// TIA Portal V17 export
// export: Created 2022-07-28T18:02:50.8696399Z, ExportSetting None, DisplayName Totally Integrated Automation Portal, DisplayVersion V17, DisplayName TIA Portal Openness, DisplayVersion V17, DisplayName TIA Portal Teamcenter Gateway, DisplayVersion V17, DisplayName TIA Portal Version Control Interface, DisplayVersion V17, DisplayName TIA Portal Test Suite Advanced, DisplayVersion V17, DisplayName SINAMICS Startdrive Advanced, DisplayVersion V17, DisplayName SINAMICS DCC, DisplayVersion V17, DisplayName SINAMICS Startdrive G130, G150, S120, S150, SINAMICS MV, S210, DisplayVersion V17, DisplayName SINAMICS Startdrive G110M, G120, G120C, G120D, G120P, G115D, DisplayVersion V17, DisplayName STEP 7 Professional, DisplayVersion V17, DisplayName SIMATIC Energy Suite, DisplayVersion V17, DisplayName STEP 7 CFC, DisplayVersion V17, DisplayName STEP 7 Safety, DisplayVersion V17, DisplayName WinCC Advanced / Unified PC, DisplayVersion V17, DisplayName SIMATIC Visualization Architect, DisplayVersion V17
FUNCTION_BLOCK "Lib_FB_AnalogFlowmeter"   // FB7, SCL
{ S7_Optimized_Access := 'TRUE' }
AUTHOR : bean
// Analog sensor functional block
// stored: AutoNumber false, MemoryReserve 100, SetENOAutomatically false
   VAR_INPUT
      I_Initialization { ExternalAccessible := 'False'; ExternalVisible := 'False'; ExternalWritable := 'False'} : Bool := FALSE;   // 1 = Restart PLC is active (First scan)
      IR_Raw { ExternalAccessible := 'False'; ExternalVisible := 'False'; ExternalWritable := 'False'} : Real;   // Sensor input
      IR_High { ExternalAccessible := 'False'; ExternalVisible := 'False'; ExternalWritable := 'False'} : Real := 27648.0;   // Max sensor input val, PLC unit
      IR_Low { ExternalAccessible := 'False'; ExternalVisible := 'False'; ExternalWritable := 'False'} : Real;   // Min sensor input val, PLC unit
      IR_Coef { ExternalAccessible := 'False'; ExternalVisible := 'False'; ExternalWritable := 'False'} : Real := 60.0;   // Coeffitient for convert flow to unit/min (t/h -> kg/min ) by dividing
      II_Mode { ExternalAccessible := 'False'; ExternalVisible := 'False'; ExternalWritable := 'False'} : Int := -1;   // 0 - analog;
      I_GlobalRST { ExternalAccessible := 'False'; ExternalVisible := 'False'; ExternalWritable := 'False'} : Bool;   // Reset faults
      I_Puls_1s { ExternalAccessible := 'False'; ExternalVisible := 'False'; ExternalWritable := 'False'} : Bool;   // 1 = Once per 1 sec
      IR_CycleTime { ExternalAccessible := 'False'; ExternalVisible := 'False'; ExternalWritable := 'False'} : Real;   // PLC last cycle time
      II_Obj_ID { ExternalAccessible := 'False'; ExternalVisible := 'False'; ExternalWritable := 'False'} : Int := -1;   // Tech ID of object
   END_VAR
   VAR_OUTPUT
      QR_ScalledVal { ExternalAccessible := 'False'; ExternalVisible := 'False'; ExternalWritable := 'False'} : Real;   // Output scaled sensor value
      Q_HH { ExternalAccessible := 'False'; ExternalVisible := 'False'; ExternalWritable := 'False'} : Bool;   // High level Alarm
      Q_H { ExternalAccessible := 'False'; ExternalVisible := 'False'; ExternalWritable := 'False'} : Bool;   // High level Warning
      Q_L { ExternalAccessible := 'False'; ExternalVisible := 'False'; ExternalWritable := 'False'} : Bool;   // Low level Warning
      Q_LL { ExternalAccessible := 'False'; ExternalVisible := 'False'; ExternalWritable := 'False'} : Bool;   // Low level Alarm
      Q_Overshoot { ExternalAccessible := 'False'; ExternalVisible := 'False'; ExternalWritable := 'False'} : Bool;   // Sensor value overshoot
      Q_BadSensor { ExternalAccessible := 'False'; ExternalVisible := 'False'; ExternalWritable := 'False'} : Bool;   // Sensor in zero
      Q_DBReadErr { ExternalAccessible := 'False'; ExternalVisible := 'False'; ExternalWritable := 'False'} : Bool;   // Object DB reading fault
   END_VAR
   VAR_IN_OUT
      IQ_PLC_CycleInfo : Variant;
   END_VAR
   VAR
      s_SimMode { ExternalAccessible := 'False'; ExternalVisible := 'False'; ExternalWritable := 'False'} : Bool;   // Simulation mode is active
      s_FltCondition_HH { ExternalAccessible := 'False'; ExternalVisible := 'False'; ExternalWritable := 'False'} : Bool;   // Condition for high level fault
      s_FltCondition_H { ExternalAccessible := 'False'; ExternalVisible := 'False'; ExternalWritable := 'False'} : Bool;   // Condition for high level warning
      s_FltCondition_L { ExternalAccessible := 'False'; ExternalVisible := 'False'; ExternalWritable := 'False'} : Bool;   // Condition for low level warning
      s_FltCondition_LL { ExternalAccessible := 'False'; ExternalVisible := 'False'; ExternalWritable := 'False'} : Bool;   // Condition for low level fault
      s_Flt_HH { ExternalAccessible := 'False'; ExternalVisible := 'False'; ExternalWritable := 'False'} : Bool;
      s_Flt_LL { ExternalAccessible := 'False'; ExternalVisible := 'False'; ExternalWritable := 'False'} : Bool;
      slr_CurrentFlow_u_s { ExternalAccessible := 'False'; ExternalVisible := 'False'; ExternalWritable := 'False'} : LReal;   // Current flow in unit/sec
      slr_PrevFlow_u_s { ExternalAccessible := 'False'; ExternalVisible := 'False'; ExternalWritable := 'False'} : LReal;   // Previous flow in unit/sec
      slr_CountFlow_min { ExternalAccessible := 'False'; ExternalVisible := 'False'; ExternalWritable := 'False'} : LReal;
      slr_FlowMid_min { ExternalAccessible := 'False'; ExternalVisible := 'False'; ExternalWritable := 'False'} : LReal;
      si_CountTimePoints { ExternalAccessible := 'False'; ExternalVisible := 'False'; ExternalWritable := 'False'} : Int;
      slr_Count_unit { ExternalAccessible := 'False'; ExternalVisible := 'False'; ExternalWritable := 'False'} : LReal;   // Counter for units
      s_Enable { ExternalAccessible := 'False'; ExternalVisible := 'False'; ExternalWritable := 'False'} : Struct   // Enable/disable faults detection
         HH : Bool := true;   // High fault
         H : Bool := true;   // High warning
         L : Bool := true;   // Low warning
         LL : Bool := true;   // Low fault
      END_STRUCT;
      s_Suppressed { ExternalAccessible := 'False'; ExternalVisible := 'False'; ExternalWritable := 'False'} : Struct   // Suppress faults
         HH : Bool;   // High fault
         H : Bool;   // High warning
         L : Bool;   // Low warning
         LL : Bool;   // Low fault
      END_STRUCT;
      s_TON_HH { ExternalAccessible := 'False'; ExternalVisible := 'False'; ExternalWritable := 'False'} : "Lib_FB_Timer_ON_Simple";
      s_TON_H { ExternalAccessible := 'False'; ExternalVisible := 'False'; ExternalWritable := 'False'} : "Lib_FB_Timer_ON_Simple";
      s_TON_L { ExternalAccessible := 'False'; ExternalVisible := 'False'; ExternalWritable := 'False'} : "Lib_FB_Timer_ON_Simple";
      s_TON_LL { ExternalAccessible := 'False'; ExternalVisible := 'False'; ExternalWritable := 'False'} : "Lib_FB_Timer_ON_Simple";
      s_EdgeError { ExternalAccessible := 'False'; ExternalVisible := 'False'; ExternalWritable := 'False'} : "Lib_FB_Edge";
      s_EdgeWarning { ExternalAccessible := 'False'; ExternalVisible := 'False'; ExternalWritable := 'False'} : "Lib_FB_Edge";
      s_EdgeOvershot { ExternalAccessible := 'False'; ExternalVisible := 'False'; ExternalWritable := 'False'} : "Lib_FB_Edge";
   END_VAR
   VAR RETAIN
      s_Simulation { ExternalAccessible := 'False'; ExternalVisible := 'False'; ExternalWritable := 'False'} : Struct
         Obj_DATA_BACKUP : Struct
            Config : "_AnalogFlowmeter_Config";
            s_Enable : Struct   // Enable/disable faults detection
               HH : Bool := true;   // High fault
               H : Bool := true;   // High warning
               L : Bool := true;   // Low warning
               LL : Bool := true;   // Low fault
            END_STRUCT;
            s_Suppressed : Struct   // Suppress faults
               HH : Bool;   // High fault
               H : Bool;   // High warning
               L : Bool;   // Low warning
               LL : Bool;   // Low fault
            END_STRUCT;
         END_STRUCT;
      END_STRUCT;
      s_Obj_Retain_BUp { ExternalAccessible := 'False'; ExternalVisible := 'False'; ExternalWritable := 'False'} : Struct
         Config : "_AnalogFlowmeter_Config";
         s_Enable : Struct   // Enable/disable faults detection
            HH : Bool := true;   // High fault
            H : Bool := true;   // High warning
            L : Bool := true;   // Low warning
            LL : Bool := true;   // Low fault
         END_STRUCT;
         s_Suppressed : Struct   // Suppress faults
            HH : Bool;   // High fault
            H : Bool;   // High warning
            L : Bool;   // Low warning
            LL : Bool;   // Low fault
         END_STRUCT;
      END_STRUCT;
   END_VAR
   VAR_TEMP
      t_SomeFault : Bool;
      t_SomeWarning : Bool;
      t_SensorOvershoot : Bool;
      t_Flt_HH : Bool;
      t_Flt_H : Bool;
      t_Flt_L : Bool;
      t_Flt_LL : Bool;
      t_Flt_SensMax : Bool;
      t_Flt_SensMin : Bool;
      t_ExclFlt : Bool;   // Excluded (suppressed) fault is active
      t_RST_FLT : Bool;
      t_DBReadErr : Bool;   // Fault while DB reading
      t_ResetCurrCnt : Bool;   // 1 = Reset current counter
      t_ResetGenCnt : Bool;   // 1 = Reset general counter
      ti_DBReadErr : Int;   // Fault # while DB reading
      ti_CMDLogic : Int;   // Command word for logic
      tlr_CntLastCycle : LReal;   // Counter by last cycle, unit
      t_WholeRange : Bool;
      t_WholeRangeP : Bool;
      ti_NumObjDB : UInt;   // Number of DB for storage object data
      t_ObjAny_HMI : DB_ANY;   // Ref to object data
      t_ObjVar_HMI : Variant;   // Ref to object data
      t_ObjAny_PLC : DB_ANY;   // Ref to object data
      t_ObjVar_PLC : Variant;   // Ref to object data
      tr_OutVal : Real;   // Output Sensor Value
      tr_OutValSens : Real;   // Output value in sensor range
      tr_OutValSensProc : Real;   // Output value in sensor range in %
      tr_CurrMaxRange : Real;   // Current maxixmum value of the range
      tr_CurrMinRange : Real;   // Current minimum value of the range
      tr_SP_HH : Real;
      tr_SP_H : Real;
      tr_SP_L : Real;
      tr_SP_LL : Real;
      tr_DeltaFlt : Real;
      tr_SensorVal : Real;
      tlr_Frac_CntU : LReal;   // Frac from unit counter
      tlr_CoefChecked : LReal;
      tui_IntPart_CntU : UDInt;   // Integer part from unit counter
      td_DB_ShiftHMI : DInt;   // Object DB number shift
      td_DB_ShiftPLC : DInt;   // Object DB number shift
      t_PLC_CycleInfo : "Lib_PLC_CycleInfo";
      t_Obj_HMI : "lib_udt_AnalogFlowmeter_HMI";
      t_Obj_PLC : "lib_udt_AnalogFlowmeter_PLC";
      t_InternalData : "Lib_UDT_Int";   // Internal data
   END_VAR
BEGIN
   REGION Inputs
       //Global reset to logic
       #t_RST_FLT := #I_GlobalRST;

       //Set internal data
       REGION Internal data
           #t_InternalData.AlwTrue := true;
           #t_InternalData.AlwFalse := false;
           #t_InternalData.i_Alw0 := 0;
           #t_InternalData.b_Alw0 := b#16#0;
           #t_InternalData.w_Alw0 := w#16#0;
           #t_InternalData.d_Alw0 := dw#16#0;
       END_REGION

       //Reinit tempory variables
       REGION Reinit tempory variables
           #t_WholeRange := false;
           #t_WholeRangeP := false;
           #t_ResetCurrCnt := false;
           #t_ResetGenCnt := false;
           #tr_SP_HH := 90.0;
           #tr_SP_H := 80.0;
           #tr_SP_L := 20.0;
           #tr_SP_LL := 10.0;
           #tr_DeltaFlt := 2.0;

       END_REGION

       //Read data  PLC 
       VariantGet(SRC := #IQ_PLC_CycleInfo,
                  DST => #t_PLC_CycleInfo);

       //Read Object data
       //Reinit temp values
       #t_Obj_HMI := "D_ZeroTypes".AnalogFlowmeter_HMI;
       #t_Obj_PLC := "D_ZeroTypes".AnalogFlowmeter_PLC;
       #td_DB_ShiftHMI := "D_General_ProgramDATA".ui_Shift_DBSens_HMI;
       #td_DB_ShiftPLC := "D_General_ProgramDATA".ui_Shift_DBSens_PLC;

       IF #II_Obj_ID >= 0
       THEN
           //Read HMI data
           #ti_NumObjDB := DINT_TO_UINT(INT_TO_DINT(#II_Obj_ID) + #td_DB_ShiftHMI);
           #t_ObjAny_HMI := UINT_TO_DB_ANY(#ti_NumObjDB);
           #t_ObjVar_HMI := DB_ANY_TO_VARIANT(in := #t_ObjAny_HMI, err => #ti_DBReadErr);

           //If DB exist and convertion without error
           IF #ti_DBReadErr = 0
           THEN
               VariantGet(SRC := #t_ObjVar_HMI,
                          DST => #t_Obj_HMI);
           ELSE
               #t_DBReadErr := true;
           END_IF;

           //Read PLC data
           #ti_NumObjDB := DINT_TO_UINT(INT_TO_DINT(#II_Obj_ID) + #td_DB_ShiftPLC);
           #t_ObjAny_PLC := UINT_TO_DB_ANY(#ti_NumObjDB);
           #t_ObjVar_PLC := DB_ANY_TO_VARIANT(in := #t_ObjAny_PLC, err => #ti_DBReadErr);

           //If DB exist and convertion without error
           IF #ti_DBReadErr = 0
           THEN
               VariantGet(SRC := #t_ObjVar_PLC,
                          DST => #t_Obj_PLC);
           ELSE
               #t_DBReadErr := true;
           END_IF;
       ELSE
           #t_DBReadErr := true;
       END_IF;

       //Read retain data if initialization is active
       IF #I_Initialization
       THEN
           #t_Obj_HMI.Config := #s_Obj_Retain_BUp.Config;
           #s_Enable := #s_Obj_Retain_BUp.s_Enable;
           #s_Suppressed := #s_Obj_Retain_BUp.s_Suppressed;

           #slr_PrevFlow_u_s := 0.0;
           #slr_Count_unit := 0.0;
           #slr_CountFlow_min := 0.0;
           #slr_FlowMid_min := 0.0;
           #si_CountTimePoints := 0;
       END_IF;

       //Define CMD by priority
       IF #t_PLC_CycleInfo.CMD_GLOBAL <> 0
       THEN
           #ti_CMDLogic := #t_PLC_CycleInfo.CMD_GLOBAL;
       ELSE
           IF #t_Obj_HMI.CMD <> 0
           THEN
               #ti_CMDLogic := #t_Obj_HMI.CMD;
               #t_Obj_HMI.CMD := 0;
           END_IF;
       END_IF;

       CASE #ti_CMDLogic OF
           0:  //Do nothing
               ;
           7:  //Sim mode ON
               IF NOT #s_SimMode
               THEN
                   #s_SimMode := TRUE;
                   #s_Simulation.Obj_DATA_BACKUP.Config := #t_Obj_HMI.Config;
                   #s_Simulation.Obj_DATA_BACKUP.s_Enable := #s_Enable;
                   #s_Simulation.Obj_DATA_BACKUP.s_Suppressed := #s_Suppressed;
               END_IF;

           8:  //Sim mode OFF
               IF #s_SimMode
               THEN
                   #s_SimMode := FALSE;
                   #t_Obj_HMI.Config := #s_Simulation.Obj_DATA_BACKUP.Config;
                   #s_Enable := #s_Simulation.Obj_DATA_BACKUP.s_Enable;
                   #s_Suppressed := #s_Simulation.Obj_DATA_BACKUP.s_Suppressed;
               END_IF;

           31..32://Reset faults
               #t_RST_FLT := TRUE;
           76:  //Display whole range
               #t_Obj_HMI.Config.i_HMI_SensValRange := 0;
           77:  //Display whole range, %
               #t_Obj_HMI.Config.i_HMI_SensValRange := 1;
               (* IF #II_Mode <> 0 THEN
                   #t_Obj_HMI.Config.i_HMI_SensValRange := 1;
               ELSE
                   #t_Obj_HMI.Config.i_HMI_SensValRange := 0;
               END_IF; *)(*
           78:  //Display a part of range
               #t_Obj_HMI.Config.i_HMI_SensValRange := 2;
           79:  //Display a part of range, %
               #t_Obj_HMI.Config.i_HMI_SensValRange := 3; *)
           60: //HH fault enable / disable
               #s_Enable.HH := NOT #s_Enable.HH;
           61: //H fault enable / disable
               #s_Enable.H := NOT #s_Enable.H;
           62: //L fault enable / disable
               #s_Enable.L := NOT #s_Enable.L;
           63: //LL fault enable / disable
               #s_Enable.LL := NOT #s_Enable.LL;
           64: //HH fault suppressed / consider
               #s_Suppressed.HH := NOT #s_Suppressed.HH;
           65: //H fault suppressed / consider
               #s_Suppressed.H := NOT #s_Suppressed.H;
           66: //L fault suppressed / consider
               #s_Suppressed.L := NOT #s_Suppressed.L;
           67: //LL fault suppressed / consider
               #s_Suppressed.LL := NOT #s_Suppressed.LL;
           500: //Reset current counter
               #t_ResetCurrCnt := true;
           501: //Reset general counter
               #t_ResetGenCnt := true;
           ELSE//
               ;
       END_CASE;

       CASE #t_Obj_HMI.Config.i_HMI_SensValRange OF
           0..1:  //Valid range
               ;
           ELSE  //Invalid range
               #t_Obj_HMI.Config.i_HMI_SensValRange := 1;
       END_CASE;

       #tr_SensorVal := #IR_Raw;
   END_REGION

   REGION Min/max values check
       //Start reading limits, offset and setpoints --------limits-offset-setpoints--------limits-offset-setpoints
       //            ************
       IF #t_Obj_HMI.Config.r_MinVal > #t_Obj_HMI.Config.r_MaxVal THEN
           #t_Obj_HMI.Config.r_MinVal := #t_Obj_HMI.Config.r_MaxVal;
       END_IF;
   END_REGION

   REGION Calculate percentage value depending on the mode of the sensor

       CASE #II_Mode OF
           0:  //Analog input like 0 - 27648 -> 0 - 75 C
               IF (#IR_High - #IR_Low) <> 0.0
               THEN
                   #tr_OutValSensProc := (#tr_SensorVal - #IR_Low) / (#IR_High - #IR_Low) * 100.0;
               ELSE
                   #tr_OutValSensProc := 0.0;
               END_IF;

           ELSE  //Undefined or unchoiced type of the sensor
               #t_Obj_HMI := "D_ZeroTypes".AnalogFlowmeter_HMI;
               #t_Obj_PLC := "D_ZeroTypes".AnalogFlowmeter_PLC;

               //Write Object data
               //DB num 
               IF #II_Obj_ID >= 0
                   AND NOT #t_DBReadErr
               THEN
                   //Write HMI data
                   VariantPut(SRC := #t_Obj_HMI,
                              DST := #t_ObjVar_HMI);

                   //Write PLC data
                   VariantPut(SRC := #t_Obj_PLC,
                              DST := #t_ObjVar_PLC);
               ELSE
                   #t_DBReadErr := true;
               END_IF;

               #QR_ScalledVal := 0.0;
               #Q_HH :=
               #Q_H :=
               #Q_L :=
               #Q_LL :=
               #Q_Overshoot :=
               #Q_DBReadErr := false;

               RETURN;
       END_CASE;

       //Calculate all others out values
       #tr_OutValSens := (#t_Obj_HMI.Config.r_MaxVal - #t_Obj_HMI.Config.r_MinVal) * #tr_OutValSensProc / 100.0 + #t_Obj_HMI.Config.r_MinVal;

       //Assign display mode depending by display mode
       CASE #t_Obj_HMI.Config.i_HMI_SensValRange OF
           0: //Display whole range
               #tr_OutVal := #tr_OutValSens + #t_Obj_HMI.Config.r_Offset;
               #tr_CurrMaxRange := #t_Obj_HMI.Config.r_MaxVal;
               #tr_CurrMinRange := #t_Obj_HMI.Config.r_MinVal;
               #t_WholeRange := true;
           1: //Display whole range (percents)
               #tr_OutVal := #tr_OutValSensProc + #t_Obj_HMI.Config.r_Offset;
               #tr_CurrMaxRange := 100.0;
               #tr_CurrMinRange := 0.0;
               #t_WholeRangeP := true;
           ELSE
               ;
       END_CASE;

       REGION Check limits, zero of sensor ect.
           IF #tr_SensorVal < #IR_Low
               OR #tr_SensorVal > #IR_High
           THEN
               #t_SensorOvershoot := true;
           END_IF;

           IF #tr_OutValSensProc < -5.0
           THEN
               #t_Flt_SensMin := TRUE;
               #tr_OutVal := 0.0;
           END_IF;

           IF #tr_OutValSensProc > 105.0
           THEN
               #t_Flt_SensMax := TRUE;
               #tr_OutVal := 0.0;
           END_IF;

           IF #tr_OutVal > #tr_CurrMaxRange
           THEN
               #tr_OutVal := #tr_CurrMaxRange;
           END_IF;
           IF #tr_OutVal < #tr_CurrMinRange
           THEN
               #tr_OutVal := #tr_CurrMinRange;
           END_IF;
       END_REGION

       IF #s_SimMode
       THEN
           #tr_OutVal := #t_Obj_HMI.Config.r_DisplayData;
           #tr_OutValSens := #t_Obj_HMI.Config.r_DisplayData;
       END_IF;

   END_REGION

   REGION Calculate counters by flow
       //Reset counters
       IF #t_ResetCurrCnt
       THEN
           #t_Obj_HMI.Config.r_CountCurr := 0;
       END_IF;
       IF #t_ResetGenCnt
       THEN
           #t_Obj_HMI.Config.r_CountGen := 0;
       END_IF;

       IF #I_Puls_1s
       THEN

           //Check coeffitient
           IF #IR_Coef <> 0.0
           THEN
               #tlr_CoefChecked := REAL_TO_LREAL(#IR_Coef);
           ELSE
               #tlr_CoefChecked := 1.0;
           END_IF;

           //Calculate counter by previous cycle
           #slr_CurrentFlow_u_s := REAL_TO_LREAL(#tr_OutValSens) / #tlr_CoefChecked;

           //Count time points and sum of flow
           #slr_CountFlow_min += #slr_CurrentFlow_u_s;
           #si_CountTimePoints += 1;

           IF #si_CountTimePoints >= 60
           THEN
               #slr_FlowMid_min += #slr_CountFlow_min / 60.0;

               #si_CountTimePoints := 0;

               #tui_IntPart_CntU := DINT_TO_UDINT(TRUNC(#slr_FlowMid_min));
               #tlr_Frac_CntU := FRAC(#slr_FlowMid_min);
               #slr_CountFlow_min := 0.0;//#tlr_Frac_CntU;
               #slr_FlowMid_min := #tlr_Frac_CntU;

               #t_Obj_HMI.Config.r_CountCurr += #tui_IntPart_CntU;
               #t_Obj_HMI.Config.r_CountGen += #tui_IntPart_CntU;
               #t_Obj_HMI.Config.r_CountHour += #tui_IntPart_CntU;
           END_IF;

       END_IF;


   END_REGION

   REGION Setpoints values check
       //            ************
       IF #t_Obj_HMI.Config.r_LL_Setpoint < #tr_CurrMinRange
       THEN
           #t_Obj_HMI.Config.r_LL_Setpoint := #tr_CurrMinRange;
       ELSIF #t_Obj_HMI.Config.r_LL_Setpoint > #tr_CurrMaxRange
       THEN
           #t_Obj_HMI.Config.r_LL_Setpoint := #tr_CurrMaxRange;
       END_IF;

       IF #t_Obj_HMI.Config.r_HH_Setpoint > #tr_CurrMaxRange
       THEN
           #t_Obj_HMI.Config.r_HH_Setpoint := #tr_CurrMaxRange;
       ELSIF #t_Obj_HMI.Config.r_HH_Setpoint < #tr_CurrMinRange
       THEN
           #t_Obj_HMI.Config.r_HH_Setpoint := #tr_CurrMinRange;
       END_IF;
       //            ************
       IF #t_Obj_HMI.Config.r_H_Setpoint > #t_Obj_HMI.Config.r_HH_Setpoint
       THEN
           #t_Obj_HMI.Config.r_H_Setpoint := #t_Obj_HMI.Config.r_HH_Setpoint;
       ELSIF #t_Obj_HMI.Config.r_H_Setpoint < #t_Obj_HMI.Config.r_LL_Setpoint
       THEN
           #t_Obj_HMI.Config.r_H_Setpoint := #t_Obj_HMI.Config.r_LL_Setpoint;
       END_IF;

       IF #t_Obj_HMI.Config.r_L_Setpoint > #t_Obj_HMI.Config.r_H_Setpoint
       THEN
           #t_Obj_HMI.Config.r_L_Setpoint := #t_Obj_HMI.Config.r_H_Setpoint;
       ELSIF #t_Obj_HMI.Config.r_L_Setpoint < #t_Obj_HMI.Config.r_LL_Setpoint
       THEN
           #t_Obj_HMI.Config.r_L_Setpoint := #t_Obj_HMI.Config.r_LL_Setpoint;
       END_IF;

       //            ************         
       #tr_SP_HH := #t_Obj_HMI.Config.r_HH_Setpoint;
       #tr_SP_H := #t_Obj_HMI.Config.r_H_Setpoint;
       #tr_SP_L := #t_Obj_HMI.Config.r_L_Setpoint;
       #tr_SP_LL := #t_Obj_HMI.Config.r_LL_Setpoint;
       #tr_DeltaFlt := #t_Obj_HMI.Config.r_Hysteresis;
       //Finish reading limits, offset and setpoints --------limits-offset-setpoints--------limits-offset-setpoints
   END_REGION

   REGION Warnings AND faults

       REGION Setpoints intersection    
           //Setpoints intersection
           IF #tr_SP_HH <= #tr_CurrMaxRange
               AND #tr_SP_H <= #tr_CurrMaxRange
           THEN
               #s_FltCondition_HH := (#tr_SP_HH <= #tr_OutVal)
               OR (#s_FltCondition_HH
               AND #tr_OutVal >= (#tr_SP_HH - #tr_DeltaFlt));

               #s_FltCondition_H := (#tr_SP_H <= #tr_OutVal)
               OR (#s_FltCondition_H
               AND #tr_OutVal >= (#tr_SP_H - #tr_DeltaFlt));

           ELSE
               #s_FltCondition_HH := FALSE;
               #s_FltCondition_H := FALSE;
           END_IF;

           IF #tr_SP_LL >=  #tr_CurrMinRange
               AND #tr_SP_L >= #tr_CurrMinRange
           THEN
               #s_FltCondition_LL := (#tr_SP_LL >= #tr_OutVal)
               OR (#s_FltCondition_LL
               AND #tr_OutVal <= (#tr_SP_LL + #tr_DeltaFlt));

               #s_FltCondition_L := (#tr_SP_L >= #tr_OutVal)
               OR (#s_FltCondition_L
               AND #tr_OutVal <= (#tr_SP_L + #tr_DeltaFlt));
           ELSE
               #s_FltCondition_LL := FALSE;
               #s_FltCondition_L := FALSE;
           END_IF;
       END_REGION

       //Enabled faults and warnings check
       #s_FltCondition_HH := #s_FltCondition_HH AND #s_Enable.HH;
       #s_FltCondition_H := #s_FltCondition_H AND #s_Enable.H;
       #s_FltCondition_L := #s_FltCondition_L AND #s_Enable.L;
       #s_FltCondition_LL := #s_FltCondition_LL AND #s_Enable.LL;

       #s_TON_HH(IB_StartTimerInput := #s_FltCondition_HH,
               IR_CycleTime := #IR_CycleTime,
               IR_SpTime := #t_Obj_HMI.Config.r_WarnDetectTime);

       #s_TON_H(IB_StartTimerInput := #s_FltCondition_H,
              IR_CycleTime := #IR_CycleTime,
              IR_SpTime := #t_Obj_HMI.Config.r_WarnDetectTime);

       #s_TON_L(IB_StartTimerInput := #s_FltCondition_L,
              IR_CycleTime := #IR_CycleTime,
              IR_SpTime := #t_Obj_HMI.Config.r_WarnDetectTime);

       #s_TON_LL(IB_StartTimerInput := #s_FltCondition_LL,
               IR_CycleTime := #IR_CycleTime,
               IR_SpTime := #t_Obj_HMI.Config.r_WarnDetectTime);

       #t_Flt_HH := #s_TON_HH.QB_TimerOut AND NOT #s_Suppressed.HH;
       #t_Flt_H := #s_TON_H.QB_TimerOut AND NOT #s_Suppressed.H;
       #t_Flt_L := #s_TON_L.QB_TimerOut AND NOT #s_Suppressed.L;
       #t_Flt_LL := #s_TON_LL.QB_TimerOut AND NOT #s_Suppressed.LL;

       //Excluded (suppressed) fault is active
       #t_ExclFlt := (#s_TON_HH.QB_TimerOut AND #s_Suppressed.HH)
       OR (#s_TON_H.QB_TimerOut AND #s_Suppressed.H)
       OR (#s_TON_L.QB_TimerOut AND #s_Suppressed.L)
       OR (#s_TON_LL.QB_TimerOut AND #s_Suppressed.LL)
       ;

       #s_Flt_HH := #t_Flt_HH
       OR (#s_Flt_HH
       AND NOT #t_RST_FLT);

       #s_Flt_LL := #t_Flt_LL
       OR (#s_Flt_LL
       AND NOT #t_RST_FLT);


       //Some fault is active
       #t_SomeFault := #s_Flt_HH
       OR #s_Flt_LL
       ;
       //Some warning is active
       #t_SomeWarning := #t_Flt_H
       OR #t_Flt_L
       ;
       //New fault checking
       #s_EdgeError(IB_Input := #t_SomeFault);

       //New warning checking
       #s_EdgeWarning(IB_Input := #t_SomeWarning);

       //New overshot detected
       #s_EdgeOvershot(IB_Input := #t_SensorOvershoot
                       OR #t_Flt_SensMax
                       OR #t_Flt_SensMin);
   END_REGION

   REGION PLC State + Counter
       "Lib_FC_ASens_CycleInfo_Count_State"(Alarm := #t_SomeFault,
                                            AlarmNew := #s_EdgeError.QB_EdgePos,
                                            Warning := #t_SomeWarning,
                                            WarningNew := #s_EdgeWarning.QB_EdgePos,

                                            ErrorBad := #t_SensorOvershoot
                                            OR #t_Flt_SensMax
                                            OR #t_Flt_SensMin,
                                            ErrorBadNew := #s_EdgeOvershot.QB_EdgePos,
                                            Simulation := #s_SimMode,
                                            PLC_CycleInfo := #t_PLC_CycleInfo);
   END_REGION

   REGION BUp Data
       IF NOT #I_Initialization
       THEN
           #s_Obj_Retain_BUp.Config := #t_Obj_HMI.Config;
           #s_Obj_Retain_BUp.s_Enable := #s_Enable;
           #s_Obj_Retain_BUp.s_Suppressed:= #s_Suppressed;
       END_IF;
   END_REGION

   REGION Outputs
       //Outputs
       //Object DBs
       //HMI DB
       #t_Obj_HMI.Config.r_DisplayData := #tr_OutVal;
       #t_Obj_HMI.ID := #II_Obj_ID;
       #t_Obj_HMI.CLSID := 40;
       #t_Obj_HMI.Status.r_HW_Value := #IR_Raw;

       //Alarm word
       #t_Obj_HMI.Status.w_AW1.%X0 := #s_Flt_HH;           //x0 - HH fault is active                       
       #t_Obj_HMI.Status.w_AW1.%X1 := #t_Flt_H;            //x1 - H fault is active                        
       #t_Obj_HMI.Status.w_AW1.%X2 := #t_Flt_L;            //x2 - L fault is active                        
       #t_Obj_HMI.Status.w_AW1.%X3 := #s_Flt_LL;           //x3 - LL fault is active                       
       #t_Obj_HMI.Status.w_AW1.%X4 := #t_SensorOvershoot;  //x4 - Overshoot is active (act val > Maxlim)   
       #t_Obj_HMI.Status.w_AW1.%X5 := #t_Flt_SensMax;      //x5 - Exceeding the maximum                    
       #t_Obj_HMI.Status.w_AW1.%X6 := #t_Flt_SensMin;      //x6 - Exceeding the minimum                    
       #t_Obj_HMI.Status.w_AW1.%X7 := #s_SimMode;          //x7 - Sim mode is active                       
       #t_Obj_HMI.Status.w_AW1.%X8 := NOT #s_SimMode;      //x8 - Sim mode disabled
   (*    #t_Obj_HMI.Status.w_AW1.%X9     := ;    //x9 - 
       #t_Obj_HMI.Status.w_AW1.%X10    := ;    //x10 - 
       #t_Obj_HMI.Status.w_AW1.%X11    := ;    //x11 - 
       #t_Obj_HMI.Status.w_AW1.%X12    := ;    //x12 - 
       #t_Obj_HMI.Status.w_AW1.%X13    := ;    //x13 - 
       #t_Obj_HMI.Status.w_AW1.%X14    := ;    //x14 - 
       #t_Obj_HMI.Status.w_AW1.%X15    := ;    //x15 - Not used *)

       #t_Obj_HMI.Status.w_AW2.%X0 := NOT #s_Enable.HH;        //x0 - Disable HH fault detection
       #t_Obj_HMI.Status.w_AW2.%X1 := NOT #s_Enable.H;         //x1 - Disable H fault detection   
       #t_Obj_HMI.Status.w_AW2.%X2 := NOT #s_Enable.L;         //x2 - Disable L fault detection   
       #t_Obj_HMI.Status.w_AW2.%X3 := NOT #s_Enable.LL;        //x3 - Disable LL fault detection
       #t_Obj_HMI.Status.w_AW2.%X4 := #s_Suppressed.HH;    //x4 - Suppress faults. HH  
       #t_Obj_HMI.Status.w_AW2.%X5 := #s_Suppressed.H;     //x5 - Suppress faults. H   
       #t_Obj_HMI.Status.w_AW2.%X6 := #s_Suppressed.L;     //x6 - Suppress faults. L   
       #t_Obj_HMI.Status.w_AW2.%X7 := #s_Suppressed.LL;    //x7 - Suppress faults. LL  
       #t_Obj_HMI.Status.w_AW2.%X8 := #t_WholeRange;       //x8 - Display whole range  
       #t_Obj_HMI.Status.w_AW2.%X9 := #t_WholeRangeP;      //x9 - Display whole range (percents)   
       #t_Obj_HMI.Status.w_AW2.%X10 := false;       //x10 - Display a part of range 
       #t_Obj_HMI.Status.w_AW2.%X11 := false;      //x11 - Display a part of range (percents)
   (*    #t_Obj_HMI.Status.w_AW2.%X12    := ;    //x12 - 
       #t_Obj_HMI.Status.w_AW2.%X13    := ;    //x13 - 
       #t_Obj_HMI.Status.w_AW2.%X14    := ;    //x14 - 
       #t_Obj_HMI.Status.w_AW2.%X15    := ;    //x15 - Not Used *)

       #t_Obj_HMI.Status.w_AW3.%X0 := #s_Enable.HH;            //x0 - Enable faults detection. HH  
       #t_Obj_HMI.Status.w_AW3.%X1 := #s_Enable.H;             //x1 - Enable faults detection. H   
       #t_Obj_HMI.Status.w_AW3.%X2 := #s_Enable.L;             //x2 - Enable faults detection. L   
       #t_Obj_HMI.Status.w_AW3.%X3 := #s_Enable.LL;            //x3 - Enable faults detection. LL  
       #t_Obj_HMI.Status.w_AW3.%X4 := NOT #s_Suppressed.HH;    //x4 - Consider HH fault    
       #t_Obj_HMI.Status.w_AW3.%X5 := NOT #s_Suppressed.H;     //x5 - Consider H fault 
       #t_Obj_HMI.Status.w_AW3.%X6 := NOT #s_Suppressed.L;     //x6 - Consider L fault 
       #t_Obj_HMI.Status.w_AW3.%X7 := NOT #s_Suppressed.LL;    //x7 - Consider LL fault    
   (*    #t_Obj_HMI.Status.w_AW3.%X8   := ;    //x8 - 
       #t_Obj_HMI.Status.w_AW3.%X9     := ;    //x9 - 
       #t_Obj_HMI.Status.w_AW3.%X10    := ;    //x10 - 
       #t_Obj_HMI.Status.w_AW3.%X11    := ;    //x11 - 
       #t_Obj_HMI.Status.w_AW3.%X12    := ;    //x12 - 
       #t_Obj_HMI.Status.w_AW3.%X13    := ;    //x13 - 
       #t_Obj_HMI.Status.w_AW3.%X14    := ;    //x14 - 
       #t_Obj_HMI.Status.w_AW3.%X15    := ;    //x15 - Not Used *)

       //Status word
       #t_Obj_HMI.Status.dw_STW.%X0 := #t_SomeFault;        //x0 - Some fault
       #t_Obj_HMI.Status.dw_STW.%X1 := #t_SomeWarning;      //x1 - Some warning
       #t_Obj_HMI.Status.dw_STW.%X2 := #t_ExclFlt;          //x2 - Excluded (suppressed) fault is active
       #t_Obj_HMI.Status.dw_STW.%X3 := NOT #s_Enable.HH;        //x3 - Disable HH fault detection
       #t_Obj_HMI.Status.dw_STW.%X4 := NOT #s_Enable.H;         //x4 - Disable H fault detection
       #t_Obj_HMI.Status.dw_STW.%X5 := NOT #s_Enable.L;         //x5 - Disable L fault detection
       #t_Obj_HMI.Status.dw_STW.%X6 := NOT #s_Enable.LL;        //x6 - Disable LL fault detection
       #t_Obj_HMI.Status.dw_STW.%X7 := #s_Suppressed.HH;    //x7 - Suppress faults. HH
       #t_Obj_HMI.Status.dw_STW.%X8 := #s_Suppressed.H;     //x8 - Suppress faults. H
       #t_Obj_HMI.Status.dw_STW.%X9 := #s_Suppressed.L;     //x9 - Suppress faults. L
       #t_Obj_HMI.Status.dw_STW.%X10 := #s_Suppressed.LL;   //x10 - Suppress faults. LL
       #t_Obj_HMI.Status.dw_STW.%X11 := #t_WholeRange;      //x11 - Display whole range
       #t_Obj_HMI.Status.dw_STW.%X12 := #t_WholeRangeP;     //x12 - Display whole range (percents)
       #t_Obj_HMI.Status.dw_STW.%X13 := false;       //x13 - Display a part of range
       #t_Obj_HMI.Status.dw_STW.%X14 := false;      //x14 - Display a part of range (percents)
       #t_Obj_HMI.Status.dw_STW.%X15 := #t_SensorOvershoot; //x15 - Active value outrange set limits
       #t_Obj_HMI.Status.dw_STW.%X16 := #t_Flt_SensMax OR #t_Flt_SensMin;//x16 - Sensor input data fault
   (*    #t_Obj_HMI.Status.dw_STW.%X17 := false;    //x17 - 
       #t_Obj_HMI.Status.dw_STW.%X18 := false;    //x18 - 
       #t_Obj_HMI.Status.dw_STW.%X19 := false;    //x19 - 
       #t_Obj_HMI.Status.dw_STW.%X20 := false;    //x20 - 
       #t_Obj_HMI.Status.dw_STW.%X21 := false;    //x21 - 
       #t_Obj_HMI.Status.dw_STW.%X22 := false;    //x22 - 
       #t_Obj_HMI.Status.dw_STW.%X23 := false;    //x23 -  *)
       #t_Obj_HMI.Status.dw_STW.%X24 := #s_SimMode;          //x24 - Sim mode is active
   (*    #t_Obj_HMI.Status.dw_STW.%X25 := false;    //x25 - 
       #t_Obj_HMI.Status.dw_STW.%X26 := false;    //x26 - 
       #t_Obj_HMI.Status.dw_STW.%X27 := false;    //x27 - 
       #t_Obj_HMI.Status.dw_STW.%X28 := false;    //x28 - 
       #t_Obj_HMI.Status.dw_STW.%X29 := false;    //x29 - 
       #t_Obj_HMI.Status.dw_STW.%X30 := false;    //x30 - 
       #t_Obj_HMI.Status.dw_STW.%X31 := false;    //x31 - Not used *)


       //PLC DB
       //Alarm word
       #t_Obj_PLC.Alarm.ErrorHH := #s_Flt_HH;
       #t_Obj_PLC.Alarm.ErrorH := #t_Flt_H;
       #t_Obj_PLC.Alarm.ErrorL := #t_Flt_L;
       #t_Obj_PLC.Alarm.ErrorLL := #s_Flt_LL;
       #t_Obj_PLC.Alarm.ErrorOvershoot := #t_SensorOvershoot;//Sensor Overshoot
       #t_Obj_PLC.Alarm.ErrorHiLimit := #t_Flt_SensMax;    //Exceeding the maximum
       #t_Obj_PLC.Alarm.ErrorLoLimit := #t_Flt_SensMin;    //Exceeding the minimum
       #t_Obj_PLC.Alarm.SimMode := #s_SimMode;
       #t_Obj_PLC.Alarm.NotSimMode := NOT #s_SimMode;

           //Disable fault detection
       #t_Obj_PLC.Alarm.DisableHH := NOT #s_Enable.HH;
       #t_Obj_PLC.Alarm.DisableH := NOT #s_Enable.H;
       #t_Obj_PLC.Alarm.DisableL := NOT #s_Enable.L;
       #t_Obj_PLC.Alarm.DisableLL := NOT #s_Enable.LL;

           //Suppressed faults
       #t_Obj_PLC.Alarm.SuppressedHH := #s_Suppressed.HH;
       #t_Obj_PLC.Alarm.SuppressedH := #s_Suppressed.H;
       #t_Obj_PLC.Alarm.SuppressedL := #s_Suppressed.L;
       #t_Obj_PLC.Alarm.SuppressedLL := #s_Suppressed.LL;

           //Enable fault detection
       #t_Obj_PLC.Alarm.EnableHH := #s_Enable.HH;
       #t_Obj_PLC.Alarm.EnableH := #s_Enable.H;
       #t_Obj_PLC.Alarm.EnableL := #s_Enable.L;
       #t_Obj_PLC.Alarm.EnableLL := #s_Enable.LL;

           //Consider faults
       #t_Obj_PLC.Alarm.ConsiderHH := NOT #s_Suppressed.HH;
       #t_Obj_PLC.Alarm.ConsiderH := NOT #s_Suppressed.H;
       #t_Obj_PLC.Alarm.ConsiderL := NOT #s_Suppressed.L;
       #t_Obj_PLC.Alarm.ConsiderLL := NOT #s_Suppressed.LL;

       //Status word
       #t_Obj_PLC.State.SimMode := #s_SimMode;     //Sim mode is active
       #t_Obj_PLC.State.Error := #t_SomeFault;     //Some fault is active
       #t_Obj_PLC.State.Warning := #t_SomeWarning; //Some warning is active
       #t_Obj_PLC.State.Suppresed := #t_ExclFlt;   //Excluded (suppressed) fault is active
       #t_Obj_PLC.State.ErrorBadSensor := #t_Flt_SensMax
       OR #t_Flt_SensMin;

           //Enable/disable faults detection
       #t_Obj_PLC.State.DisableHH := NOT #s_Enable.HH;
       #t_Obj_PLC.State.DisableH := NOT #s_Enable.H;
       #t_Obj_PLC.State.DisableL := NOT #s_Enable.L;
       #t_Obj_PLC.State.DisableLL := NOT #s_Enable.LL;

           //Suppress faults
       #t_Obj_PLC.State.SuppressedHH := #s_Suppressed.HH;
       #t_Obj_PLC.State.SuppressedH := #s_Suppressed.H;
       #t_Obj_PLC.State.SuppressedL := #s_Suppressed.L;
       #t_Obj_PLC.State.SuppressedLL := #s_Suppressed.LL;

           //Display data format
       #t_Obj_PLC.State.DispWholeRange := #t_WholeRange;    //Display whole range
       #t_Obj_PLC.State.DispWholPerc := #t_WholeRangeP;    //Display whole range (percents)
       #t_Obj_PLC.State.DispPartRange := false;     //Display a part of range
       #t_Obj_PLC.State.DispPartPerc := false;    //Display a part of range (percents)

   //Write Object data
   //DB num 
   IF #II_Obj_ID >= 0
       AND NOT #t_DBReadErr
   THEN
       //Write HMI data
       VariantPut(SRC := #t_Obj_HMI,
                  DST := #t_ObjVar_HMI);

       //Write PLC data
       VariantPut(SRC := #t_Obj_PLC,
                  DST := #t_ObjVar_PLC);
   ELSE
       #t_DBReadErr := true;
   END_IF;

       VariantPut(SRC := #t_PLC_CycleInfo,
                  DST := #IQ_PLC_CycleInfo);

       //Block outputs
       #Q_Overshoot := #t_SensorOvershoot;
       #Q_DBReadErr := #t_DBReadErr;

       #Q_HH := #s_Flt_HH;
       #Q_H := #t_Flt_H;
       #Q_L := #t_Flt_L;
       #Q_LL := #s_Flt_LL;

       #QR_ScalledVal := #tr_OutVal;
       #Q_BadSensor := #t_Obj_PLC.State.ErrorBadSensor;
   END_REGION
END_FUNCTION_BLOCK
